// TIA Portal V20 export
FUNCTION_BLOCK "SummarizeCommandsToUnit"   // FB25, SCL
{ S7_Optimized_Access := 'TRUE' }
// stored: IsIECCheckEnabled true, MemoryReserve 100, SetENOAutomatically true
   VAR_INPUT
      enable { ExternalAccessible := 'False'; ExternalVisible := 'False'; ExternalWritable := 'False'} : Bool := true;   // Enable block functionality
      eventCommands { ExternalAccessible := 'False'; ExternalVisible := 'False'; ExternalWritable := 'False'} : "LUC_typeStateCommands";   // Commands triggered by events. Connect events here that trigger commands without activating an alarm.
   END_VAR
   VAR_OUTPUT
      commandsToUnit { ExternalWritable := 'False'} : "LUC_typeStateCommands";   // Connect the feedbackToUnit data structure
      parentAlarmDB { ExternalWritable := 'False'} : "LAF_typeAlarms";   // Connect the parent alarm structure
      hmiInterfaceDB { ExternalWritable := 'False'} : "LAF_typeAlarms";   // Connect the HMI interface alarm structure for the EM level
      error { ExternalAccessible := 'False'; ExternalVisible := 'False'; ExternalWritable := 'False'} : Bool;   // Configuration error present
      status { ExternalAccessible := 'False'; ExternalVisible := 'False'; ExternalWritable := 'False'} : Word;   // Block status : 7000 No Call, 7002: Executing , 8200: Error - Wrong Config parameter
   END_VAR
   VAR_IN_OUT
      proDiagState : SV_FB_State_V2;   // Connect the ProDiag 'State' type; If ProDIag is not available, create and assign a dummy variable using the type 'SV_FB_State_V2'
      errors : Array[*] of "LAF_typeAlarm";   // Connect the Alarm DB Array for errors with no reaction
      warnings : Array[*] of "LAF_typeAlarm";   // Connect the Alarm DB Array for warnings with no reaction
      information : Array[*] of "LAF_typeAlarm";   // Connect the Alarm DB Array for Information Messages
      criteriaAnalysis : Array[*] of "LAF_typeAlarm";   // Connect the Alarm DB Array for Criteria Analysis messages
   END_VAR
   VAR
      statStatus { ExternalAccessible := 'False'; ExternalVisible := 'False'; ExternalWritable := 'False'} : Word;   // Static variable for the block status
      statBounds { ExternalAccessible := 'False'; ExternalVisible := 'False'; ExternalWritable := 'False'} : Struct   // Bounds for alarm arrays
         error : Struct   // error no reaction alarms array bounds
            lower : DInt;   // lower bound
            upper : DInt;   // upper bound
         END_STRUCT;
         warning : Struct   // warning no reactionvalarms array bounds
            lower : DInt;   // lower bound
            upper : DInt;   // upper bound
         END_STRUCT;
         information : Struct   // information alarms arrays bounds
            lower : DInt;   // lower bound
            upper : DInt;   // upper bound
         END_STRUCT;
         criteriaAnalysis : Struct   // citeria analysis alarms array bounds
            lower : DInt;   // lower bound
            upper : DInt;   // upper bound
         END_STRUCT;
      END_STRUCT;
      statEnableOld { ExternalAccessible := 'False'; ExternalVisible := 'False'; ExternalWritable := 'False'} : Bool;   // Previous enable state
      statError { ExternalAccessible := 'False'; ExternalVisible := 'False'; ExternalWritable := 'False'} : Bool;   // static bool that indicatesif the block has an error
   END_VAR
   VAR_TEMP
      tempIndex : DInt;   // Loop variable
      tempAlarms : "LAF_typeAlarms";
      tempCommands : "LUC_typeStateCommands";
      tempEnable : Bool;   // Temp variable to transfer the Enable input
   END_VAR
   VAR CONSTANT
      ARRAY_DIMENSION : UDInt := 1;   // Dimension of array*
      FB_STATE_NO_PROCESSING : DInt := 0;   // FB state: No processing
      FB_STATE_BLOCK_ERR : DInt := 30;   // FB state: Error in block
      STATUS_NO_CALL : Word := 16#7000;   // No job being currently processed
      STATUS_FIRST_CALL : Word := 16#7001;   // First call after incoming new job (rising edge 'enable')
      STATUS_SUBSEQUENT_CALL : Word := 16#7002;   // Subsequent call during active processing
      ERROR_PRESENT : Word := 16#8000;   // Starting range of error codes
      ERR_WRONG_PARAM : Word := 16#8200;   // Error: Wrong value in Config parameter
      NO_REACTION : UDInt := 0;
      STOP : UDInt := 1;
      CONTINUE : UDInt := 2;
      ABORT : UDInt := 3;
      HOLD : UDInt := 4;
      SUSPEND : UDInt := 5;
      RESET : UDInt := 6;
      START : UDInt := 7;
      UNHOLD : UDInt := 8;
      UNSUSPEND : UDInt := 9;
      CLEAR : UDInt := 10;
      COMPLETE : UDInt := 11;
   END_VAR
BEGIN
   REGION BLOCK INFO HEADER
       //===============================================================================
       // Siemens AG / (c)Copyright 2025
       //-------------------------------------------------------------------------------
       // Title:            LAF_DeriveCommandsFromAlarms
       // Comment/Function: This function derives commands for the Unit based on the configured Alarms. 
       // Library/Family:   Library of Automation Framework
       // Author:           Siemens Digital Industries
       // Tested with:      S7-PLCSIM  V20 
       // Engineering:      TIA Portal V20
       // Restrictions:     -
       // Requirements:     -
       //-------------------------------------------------------------------------------
       // Change log table:
       // Version  | Date       | Expert in charge        | Changes applied
       //----------|------------|-------------------------|-----------------------------
       // 01.00.00 | 31.03.2025 | SIMATIC Systems Support | First released version

       //===============================================================================
   END_REGION BLOCK INFO HEADER

   REGION DESCRIPTION
   (/*This block processes the Unit or Em alarms and, depending on the alarm type, sets the commands that modify the Unit's state.
       The block can be configured to evaluate either ProDiag alarms or Bit alarms. To do this, the config parameter has two possible values:*/)
   END_REGION DESCRIPTION

   REGION INPUTS

       // Copy input to temp variable for optimized performance
       #tempEnable := #enable;

   END_REGION INPUTS

   REGION ENABLING/DISABLING

       IF (#tempEnable = TRUE) AND (#statStatus = #STATUS_NO_CALL) THEN // First call: Initialize/ Enable function block

           // Set status output of the block
           #statError := FALSE;
           #statStatus := #STATUS_FIRST_CALL;

           // Detect lower and upper boundries of arrays
           REGION DETECT ARRAY BOUNDRIES
                   // Error array 
                   #statBounds.error.lower := LOWER_BOUND(ARR := #errors, DIM := #ARRAY_DIMENSION);
                   #statBounds.error.upper := UPPER_BOUND(ARR := #errors, DIM := #ARRAY_DIMENSION);

                   // Warning array
                   #statBounds.warning.lower := LOWER_BOUND(ARR := #warnings, DIM := #ARRAY_DIMENSION);
                   #statBounds.warning.upper := UPPER_BOUND(ARR := #warnings, DIM := #ARRAY_DIMENSION);

                   // Information array
                   #statBounds.information.lower := LOWER_BOUND(ARR := #information, DIM := #ARRAY_DIMENSION);
                   #statBounds.information.upper := UPPER_BOUND(ARR := #information, DIM := #ARRAY_DIMENSION);

                   // Ctiteria analysis array
                   #statBounds.criteriaAnalysis.lower := LOWER_BOUND(ARR := #criteriaAnalysis, DIM := #ARRAY_DIMENSION);
                   #statBounds.criteriaAnalysis.upper := UPPER_BOUND(ARR := #criteriaAnalysis, DIM := #ARRAY_DIMENSION);
               END_REGION CONFIG EVALUATION

       ELSIF (#statStatus = #STATUS_FIRST_CALL) THEN // Set status identifier of subsequent call
           #statStatus := #STATUS_SUBSEQUENT_CALL;

       ELSIF (#tempEnable = FALSE) AND (#statEnableOld = TRUE) THEN
           // Disable FB 
           #statStatus := #STATUS_NO_CALL;
       END_IF;

       #statEnableOld := #tempEnable; // Store value for edge detection in next cycle

   END_REGION ENABLING/DISABLING

   IF (#statStatus = #STATUS_NO_CALL OR #statStatus >= #ERROR_PRESENT) THEN
       // No further execution
       RETURN;
   END_IF;

   REGION EVALUATION

       // Set alarms according to active ProDiag categories
       #tempAlarms.error := #proDiagState.C1;
       #tempAlarms.warning := #proDiagState.C2;
       #tempAlarms.info := #proDiagState.C3;

       // Set commands depending on ProDiag subcatergories and events 
       #tempCommands.reset := #eventCommands.reset;
       #tempCommands.start := #eventCommands.start;
       #tempCommands.stop := #eventCommands.stop OR #proDiagState.Sub_Cat_2.%X0;
       #tempCommands.hold := #eventCommands.hold OR #proDiagState.Sub_Cat_2.%X3;
       #tempCommands.unhold := #eventCommands.unhold;
       #tempCommands.suspend := #eventCommands.suspend OR #proDiagState.Sub_Cat_2.%X4;
       #tempCommands.unsuspend := #eventCommands.unsuspend;
       #tempCommands.abort := #eventCommands.abort OR #proDiagState.Sub_Cat_2.%X2;
       #tempCommands.clear := #eventCommands.clear;
       #tempCommands.complete := #eventCommands.complete;

       // Set alarms and commands depending on active alarms from DB Alarms
       REGION Error
           // Loop through all errors and set alarms status and commands accordingly
           FOR #tempIndex := #statBounds.error.lower TO #statBounds.error.upper DO
               // Set alarm status
               #tempAlarms.error := #tempAlarms.error OR (#errors[#tempIndex].trigger);

               IF #tempAlarms.error THEN
                   // Set commands
                   #tempCommands.reset := #tempCommands.reset OR (#errors[#tempIndex].reaction = #RESET);
                   #tempCommands.start := #tempCommands.start OR (#errors[#tempIndex].reaction = #START);
                   #tempCommands.stop := #tempCommands.stop OR (#errors[#tempIndex].reaction = #STOP);
                   #tempCommands.hold := #tempCommands.hold OR (#errors[#tempIndex].reaction = #HOLD);
                   #tempCommands.unhold := #tempCommands.unhold OR (#errors[#tempIndex].reaction = #UNHOLD);
                   #tempCommands.suspend := #tempCommands.suspend OR (#errors[#tempIndex].reaction = #SUSPEND);
                   #tempCommands.unsuspend := #tempCommands.unsuspend OR (#errors[#tempIndex].reaction = #UNSUSPEND);
                   #tempCommands.abort := #tempCommands.abort OR (#errors[#tempIndex].reaction = #ABORT);
                   #tempCommands.clear := #tempCommands.clear OR (#errors[#tempIndex].reaction = #CLEAR);
                   #tempCommands.complete := #tempCommands.complete OR (#errors[#tempIndex].reaction = #COMPLETE);
               END_IF;
           END_FOR;
       END_REGION

       REGION Warning
           // Loop through all warnings and set alarms status and commands accordingly
           FOR #tempIndex := #statBounds.warning.lower TO #statBounds.warning.upper DO
               // Set alarm status
               #tempAlarms.warning := #tempAlarms.warning OR (#warnings[#tempIndex].trigger);

               IF #tempAlarms.warning THEN
                   // Set commands
                   #tempCommands.reset := #tempCommands.reset OR (#warnings[#tempIndex].reaction = #RESET);
                   #tempCommands.start := #tempCommands.start OR (#warnings[#tempIndex].reaction = #START);
                   #tempCommands.stop := #tempCommands.stop OR (#warnings[#tempIndex].reaction = #STOP);
                   #tempCommands.hold := #tempCommands.hold OR (#warnings[#tempIndex].reaction = #HOLD);
                   #tempCommands.unhold := #tempCommands.unhold OR (#warnings[#tempIndex].reaction = #UNHOLD);
                   #tempCommands.suspend := #tempCommands.suspend OR (#warnings[#tempIndex].reaction = #SUSPEND);
                   #tempCommands.unsuspend := #tempCommands.unsuspend OR (#warnings[#tempIndex].reaction = #UNSUSPEND);
                   #tempCommands.abort := #tempCommands.abort OR (#warnings[#tempIndex].reaction = #ABORT);
                   #tempCommands.clear := #tempCommands.clear OR (#warnings[#tempIndex].reaction = #CLEAR);
                   #tempCommands.complete := #tempCommands.complete OR (#warnings[#tempIndex].reaction = #COMPLETE);
               END_IF;
           END_FOR;
       END_REGION

       REGION Information
           // Loop through all information and set alarms status and commands accordingly
           FOR #tempIndex := #statBounds.information.lower TO #statBounds.information.upper DO
               // Set alarm status
               #tempAlarms.info := #tempAlarms.info OR (#information[#tempIndex].trigger);

               IF #tempAlarms.info THEN
                   // Set commands
                   #tempCommands.reset := #tempCommands.reset OR (#information[#tempIndex].reaction = #RESET);
                   #tempCommands.start := #tempCommands.start OR (#information[#tempIndex].reaction = #START);
                   #tempCommands.stop := #tempCommands.stop OR (#information[#tempIndex].reaction = #STOP);
                   #tempCommands.hold := #tempCommands.hold OR (#information[#tempIndex].reaction = #HOLD);
                   #tempCommands.unhold := #tempCommands.unhold OR (#information[#tempIndex].reaction = #UNHOLD);
                   #tempCommands.suspend := #tempCommands.suspend OR (#information[#tempIndex].reaction = #SUSPEND);
                   #tempCommands.unsuspend := #tempCommands.unsuspend OR (#information[#tempIndex].reaction = #UNSUSPEND);
                   #tempCommands.abort := #tempCommands.abort OR (#information[#tempIndex].reaction = #ABORT);
                   #tempCommands.clear := #tempCommands.clear OR (#information[#tempIndex].reaction = #CLEAR);
                   #tempCommands.complete := #tempCommands.complete OR (#information[#tempIndex].reaction = #COMPLETE);
               END_IF;
           END_FOR;
       END_REGION

       REGION CriteriaAnalysis
           // Loop through all information and set alarms status and commands accordingly
           FOR #tempIndex := #statBounds.criteriaAnalysis.lower TO #statBounds.criteriaAnalysis.upper DO
               // Set alarm status
             #tempAlarms.info := #tempAlarms.info OR (#criteriaAnalysis[#tempIndex].trigger);

             IF #tempAlarms.info THEN
               // Set commands
               #tempCommands.reset := #tempCommands.reset OR (#criteriaAnalysis[#tempIndex].reaction = #RESET);
               #tempCommands.start := #tempCommands.start OR (#criteriaAnalysis[#tempIndex].reaction = #START);
               #tempCommands.stop := #tempCommands.stop OR (#criteriaAnalysis[#tempIndex].reaction = #STOP);
               #tempCommands.hold := #tempCommands.hold OR (#criteriaAnalysis[#tempIndex].reaction = #HOLD);
               #tempCommands.unhold := #tempCommands.unhold OR (#criteriaAnalysis[#tempIndex].reaction = #UNHOLD);
               #tempCommands.suspend := #tempCommands.suspend OR (#criteriaAnalysis[#tempIndex].reaction = #SUSPEND);
               #tempCommands.unsuspend := #tempCommands.unsuspend OR (#criteriaAnalysis[#tempIndex].reaction = #UNSUSPEND);
               #tempCommands.abort := #tempCommands.abort OR (#criteriaAnalysis[#tempIndex].reaction = #ABORT);
               #tempCommands.clear := #tempCommands.clear OR (#criteriaAnalysis[#tempIndex].reaction = #CLEAR);
               #tempCommands.complete := #tempCommands.complete OR (#criteriaAnalysis[#tempIndex].reaction = #COMPLETE);
             END_IF;

           END_FOR;
       END_REGION

   END_REGION EVALUATION

   REGION OUTPUTS
       // Write block status outputs
       #error := #statError;
       #status := #statStatus;

       // Write output that send the commands to the unit
       #commandsToUnit := #tempCommands;

       // Put information in Alarm DB and HmiInterface DB
       #parentAlarmDB := #hmiInterfaceDB := #tempAlarms;
   END_REGION OUTPUTS
END_FUNCTION_BLOCK
